(*********************************** G.D S.p.A. - Technical Department ***********************************
============= PROGRAM INFO ============
FOLDER:             TBD
MACHINES INVOLVED:  TBD 

============= DESCRIPTION =============
csp main interface program

============= REVISIONS ===============
Date		Version	 	Author      	Description             
----------	-------		------------  	--------------------------------------------
2019/09/27 	0000.00	 	M.Grasso		Creation of the PRG

**********************************************************************************************************)
PROGRAM _csp_case_openFlap_lowest
VAR
END_VAR

;

END_PROGRAM

(* stored: Version 1.1.0.1, ProductVersion 3.1.4022.12
   POU _csp_case_openFlap_lowest: Id {fa7c3efd-5922-424e-baf1-a44b091041fa}, SpecialFunc None *)
